{attribute 'qualified_only'}

VAR_GLOBAL
	
	//DI
		arr_DI_1008	AT%I*:	ARRAY [1..8] OF str_EL1008 	;
		arr_DI_2819	AT%I*:	ARRAY [1..16] OF str_EL2819	;
	//AI
		arr_AI_3004	AT%I*:	ARRAY [1..4] OF str_EL3004	;
		arr_AI_3152	AT%I*:	ARRAY [1..2] OF str_EL3152	;
		arr_AI_3162	AT%I*:	ARRAY [1..2] OF str_EL3162	;
		arr_AI_3114	AT%I*:	ARRAY [1..4] OF str_EL3314	;
	//AO
		arr_AO_4008	AT%Q*:	ARRAY [1..8] OF str_EL4008	;	
END_VAR

(* stored: Version 1.1.0.1, ProductVersion 3.1.4024.15
   GVL GVL_IO: Id {db6c8deb-a77a-4346-9493-8284c97e20e2} *)
